// TIA Portal V16 export
// export: Created 2022-11-17T15:49:18.9342017Z, ExportSetting WithDefaults, DisplayName Totally Integrated Automation Portal, DisplayVersion V16 Update 6, DisplayName TIA Portal Version Control Interface, DisplayVersion V16 Update 2, DisplayName TIA Portal Openness, DisplayVersion V16 Update 6, DisplayName SINAMICS Startdrive Advanced, DisplayVersion V16 Update 5, DisplayName SINAMICS Startdrive G130, G150, S120, S150, SINAMICS MV, S210, DisplayVersion V16 Update 5, DisplayName SINAMICS Startdrive G110M, G120, G120C, G120D, G120P, G115D, DisplayVersion V16 Update 5, DisplayName STEP 7 Professional, DisplayVersion V16 Update 6, DisplayName STEP 7 Safety, DisplayVersion V16, DisplayName WinCC Advanced, DisplayVersion V16 Update 6
FUNCTION "Normalisation" : Void   // FC15, FBD
{ S7_Optimized_Access := 'TRUE' }
VERSION : 0.1
// stored: AutoNumber true, IsIECCheckEnabled false, SetENOAutomatically false, UDAEnableTagReadback false
   VAR_INPUT
      value_REAL : Real;
      normalisation : Real;
   END_VAR
   VAR_OUTPUT
      value_INT : Int;
   END_VAR
   VAR_TEMP
      temp_value_DINT : DInt;
      temp_value_REAL : Real;
   END_VAR
BEGIN

REGION Network 1
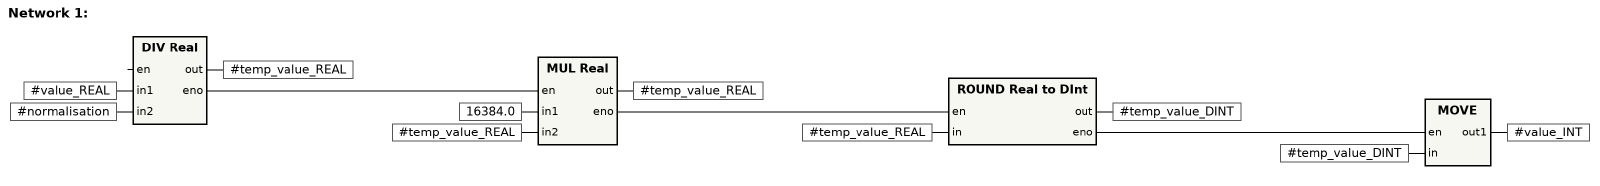
   // ENO of a box is taken as its EN; it also drops when the box reports an error
   #temp_value_REAL := #value_REAL / #normalisation;
   #temp_value_REAL := 16384.0 * #temp_value_REAL;
   #temp_value_DINT := ROUND(#temp_value_REAL);
   #value_INT := #temp_value_DINT;
END_REGION
END_FUNCTION
